INTERFACE I_Label

PROPERTY Text : STRING
GET
END_GET
SET
END_SET
END_PROPERTY

END_INTERFACE

(* stored: Version 1.1.0.1, ProductVersion 3.1.4024.12
   Itf I_Label: Id {efbe3fb4-8d6a-442e-9d7b-357fb722ddbc}
   Property Text: Id {a9dfa5f6-08b8-4212-bc0d-641b7b59fce2}
   Get Get: Id {9b65d82f-b8e4-4285-955c-62cae6cb871c}
   Set Set: Id {604d9a3c-0159-421b-baec-b593d41274ae} *)
